FUNCTION_BLOCK FB_PressureTankController EXTENDS FB_TankController
VAR_INPUT
END_VAR
VAR_OUTPUT
END_VAR
VAR
END_VAR

METHOD ControlPressure 
VAR_INPUT
END_VAR
END_METHOD

METHOD StartController
VAR_INPUT
END_VAR
SUPER^.StartController();
ControlPressure();
END_METHOD

END_FUNCTION_BLOCK

(* stored: Version 1.1.0.1, ProductVersion 3.1.4024.16
   POU FB_PressureTankController: Id {c0b4c13a-140e-4022-b223-c32a65958e4f}, SpecialFunc None
   Method ControlPressure: Id {9a6bd7d1-25c3-4fb7-9840-43f13dd7b328}
   Method StartController: Id {499e4360-ec20-4d53-945e-57af21e713b6} *)
